FUNCTION_BLOCK XtsRunner EXTENDS CyclicBase IMPLEMENTS I_XtsRunner
VAR_INPUT
END_VAR
VAR_OUTPUT
END_VAR
VAR
	CyclicModules : ARRAY[0..99] OF ICyclic;
	ModuleCount : INT := 0;
	InitModuleCount : INT := 0;
	InitialiseModules : ARRAY[0..99] OF I_Initialise;
	i: INT;
	InitialisationCount : INT;
END_VAR

METHOD AddComponent : HRESULT
VAR_INPUT
	CyclicModule : ICyclic;
END_VAR
VAR
	InitInterface : I_Initialise;
END_VAR
IF ModuleCount < 100 THEN
	CyclicModules[ModuleCount] := CyclicModule;
	IF __QUERYINTERFACE(CyclicModule,InitInterface) THEN
		InitialiseModules[ModuleCount] := InitInterface;
		InitModuleCount := InitModuleCount + 1;
	END_IF
	ModuleCount := ModuleCount + 1;
	AddComponent := 2;
ELSE
	AddComponent := S_FALSE;
END_IF
END_METHOD

METHOD Clear : HRESULT
VAR_INPUT
END_VAR
FOR i := 0 TO 99 DO
	CyclicModules[i] := 0;
	InitialiseModules[i] := 0;
END_FOR
ModuleCount := 0;
InitModuleCount := 0;
Clear := 2;
END_METHOD

METHOD PUBLIC  Cycle : HRESULT
VAR_INPUT
END_VAR
FOR i := 0 TO 99 DO
	IF CyclicModules[i] <> 0 THEN
		CyclicModules[i].Cycle();
	END_IF
END_FOR
END_METHOD

METHOD GetModuleCount : int
VAR_INPUT
END_VAR
GetModuleCount := ModuleCount;
END_METHOD

METHOD Initialise : HRESULT
VAR_INPUT
END_VAR
IF InitialisationCount < 100 THEN
	IF InitialiseModules[i] <> 0 THEN
		IF InitialiseModules[i].Initialise() = 2 THEN
			InitialisationCount := InitialisationCount + 1;
		END_IF
	ELSE
		InitialisationCount := InitialisationCount + 1;
	END_IF
ELSE
	Initialise := 2;
	InitialisationCount := 0;
END_IF
END_METHOD

METHOD RemoveModule : HRESULT
VAR_INPUT
	CyclicModule : ICyclic;
END_VAR
IF ModuleCount > 0 THEN
	RemoveModule := E_FAIL;
	FOR i := 0 TO 99 DO 
		IF CyclicModules[i] = CyclicModule THEN
			CyclicModules[i] := 0;
			IF InitialiseModules[i] <> 0 THEN
				InitialiseModules[i] := 0;
				InitModuleCount := InitModuleCount - 1;
			END_IF
			ModuleCount := ModuleCount - 1;
			RemoveModule := 2;
		END_IF
	END_FOR
ELSE
	RemoveModule := S_FALSE;
END_IF
END_METHOD

END_FUNCTION_BLOCK

(* stored: Version 1.1.0.1, ProductVersion 3.1.4024.12
   POU XtsRunner: Id {4adb75ec-914c-46a2-96a4-b49d6ed1e005}, SpecialFunc None
   Method AddComponent: Id {5f816535-6603-4c30-b42c-afe250745821}
   Method Clear: Id {801399c7-4ed5-4baa-bb84-25ca1ab9b024}
   Method Cycle: Id {07b170dc-1426-48b0-b328-82870c7027f5}
   Method GetModuleCount: Id {ce16b2d3-0e8a-4df6-aa9c-1c1b403838ba}
   Method Initialise: Id {498dbf2f-31fd-468f-af2a-ef254d08806c}
   Method RemoveModule: Id {dfa8fa7b-42f3-4591-8ff7-fdf50b44b36a} *)
